{attribute 'GeneratedUsingTerminal: EPP1322-0001-0016'}
{attribute addProperty BoxType "EPP1322-0001-0016"}
{attribute addProperty Id "InfoDataAT %I*InfoData_6F19DB2B2"}
{attribute addProperty CRC "532711307"}
{attribute addProperty Size "2"}
TYPE EPP1322_1FC0878B EXTENDS EtcSlaveTerminalBase_947E5A46 :
STRUCT
	{attribute addProperty Name "InfoData"}
	InfoData : InfoData_6F19DB2B;
END_STRUCT
END_TYPE

(* stored: Version 1.2.0.0, ProductVersion 3.1.4024.9
   DUT EPP1322_1FC0878B: Id {5f696e36-e9a8-4df1-8f2a-2b49193c0ac9} *)
